// TwinCAT 3 PLC project dmms
// ProgramVersion: 3.1.4026.18
// libraries:
//   Tc2_Standard, * (Beckhoff Automation GmbH)
//   Tc2_System, * (Beckhoff Automation GmbH)
//   Tc3_Mc3PlanarMotion, * (Beckhoff Automation GmbH)
//   Tc3_Physics, * (Beckhoff Automation GmbH)
//   Tc3_XPlanarStandard, * (Beckhoff Automation GmbH)
//   Tc3_XPlanarUtility, * (Beckhoff Automation GmbH)
// project tree:
//   / PlcTask.TcTTO
//   POUs/ FB_MotionSystem.TcPOU, MAIN.TcPOU

CONFIGURATION dmms
    RESOURCE PLC ON TwinCAT3
        TASK PlcTask(INTERVAL := T#10ms, PRIORITY := 21);
        PROGRAM MAIN WITH PlcTask : MAIN;
    END_RESOURCE
END_CONFIGURATION

// ---- POUs/MAIN.TcPOU
PROGRAM MAIN
VAR
	fbXMotionUnit : FB_MotionSystem;
	nState : UDINT;
END_VAR

CASE nState OF
	0: // Init
		nState := nState + 1;
	1: // Startup sequence
		IF fbXMotionUnit.Startup() THEN
			nState := nState + 29;
		END_IF
	30: // Preparing sequence
		IF fbXMotionUnit.Starting(bReset:= FALSE) THEN
			nState := nState + 10;
		END_IF
	40: // Executing sequence
		fbXMotionUnit.Execute(bReset:= FALSE);
END_CASE
// Cyclic update
fbXMotionUnit.Cycle();

END_PROGRAM

// ---- POUs/FB_MotionSystem.TcPOU
FUNCTION_BLOCK FB_MotionSystem
VAR
	fbXPlanarSystem : FB_XPlanarSystem;
	fbXPlanarMover  : ARRAY[1..maxNumMover] OF FB_XPlanarMoverStandard;
	nStartupSequence   : UDINT;
	nStartingSequence  : UDINT;
	nExecutingSequence : UDINT;
END_VAR

METHOD Cycle
VAR
    i : UDINT;
END_VAR
// Cyclic XPlanar objects update
fbXPlanarSystem.Cycle();
FOR i := 1 TO moverCount DO
fbXPlanarMover[i].Cycle();
END_FOR
END_METHOD

METHOD Execute : BOOL
VAR_INPUT
	bReset : BOOL; // Reset sequence
END_VAR
VAR
	i : UDINT;
END_VAR
VAR_INST
	targetPos    : ARRAY[1..maxNumMover] OF PositionXYC;
	bMoversInPos : BOOL;
	bMoverError  : BOOL;
END_VAR
IF bReset THEN
	Execute := FALSE;
	nExecutingSequence := 0;
END_IF

CASE nExecutingSequence OF
	0: // Init
		bMoversInPos := FALSE;
		bMoverError := FALSE;
		IF NOT bReset THEN
			IF fbXPlanarMover[1].P_CommandMode = MC_PLANAR_MOVER_COMMAND_MODE.FreeMovement THEN
				nExecutingSequence := nExecutingSequence + 10;
			END_IF
		END_IF

	10: // Mover 1 -> X120 Y120, Mover 2 -> X360 Y600, 500 mm/s
		targetPos[1].SetValuesXYC(120, 120, 0);
		targetPos[2].SetValuesXYC(360, 600, 0);
		FOR i := 1 TO moverCount DO
			fbXPlanarMover[i].MoveToPosition('Move to XY', targetPos[i], 500, 1250, 1250, 12500);
		END_FOR
		nExecutingSequence := nExecutingSequence + 1;

	11: // Movers moving
		bMoversInPos := TRUE;
		bMoverError := FALSE;
		FOR i := 1 TO moverCount DO
			bMoversInPos := bMoversInPos AND fbXPlanarMover[i].P_MoveToPosition.Done;
			bMoverError  := bMoverError  OR  fbXPlanarMover[i].P_MoveToPosition.Error;
		END_FOR
		IF bMoversInPos THEN
			nExecutingSequence := nExecutingSequence + 9;
		ELSIF bMoverError THEN
			nExecutingSequence := nExecutingSequence + 4;
		END_IF

	20: // Mover 1 -> X120 Y600, Mover 2 -> X360 Y120, 500 mm/s
		targetPos[1].SetValuesXYC(120, 600, 0);
		targetPos[2].SetValuesXYC(360, 120, 0);
		FOR i := 1 TO moverCount DO
			fbXPlanarMover[i].MoveToPosition('Move to XY', targetPos[i], 500, 1250, 1250, 12500);
		END_FOR
		nExecutingSequence := nExecutingSequence + 1;

	21: // Movers moving
		bMoversInPos := TRUE;
		bMoverError := FALSE;
		FOR i := 1 TO moverCount DO
			bMoversInPos := bMoversInPos AND fbXPlanarMover[i].P_MoveToPosition.Done;
			bMoverError  := bMoverError  OR  fbXPlanarMover[i].P_MoveToPosition.Error;
		END_FOR
		IF bMoversInPos THEN
			nExecutingSequence := nExecutingSequence + 9;
		ELSIF bMoverError THEN
			nExecutingSequence := nExecutingSequence + 4;
		END_IF

	30: // Done - loop
		Execute := FALSE; // operator przerywa ręcznie (Stop / E-Stop)
		nExecutingSequence := nExecutingSequence - 20; // wraca do 10 - pętla
END_CASE
END_METHOD

METHOD Starting : BOOL
VAR_INPUT
	bReset : BOOL;
END_VAR
VAR
	i : UDINT;
END_VAR
VAR_INST
	// --- diagnostyka bledu enable ---
	nErrorID       : UDINT;    // surowy kod bledu
	sErrorHex      : STRING;   // ten sam kod w HEX (do szukania w InfoSys)
	nErrObjType    : UDINT;    // typ obiektu, ktory zawinil
	nErrObjID      : UDINT;    // ktory konkretnie (np. mover 2)
	stStartCheck   : ARRAY[1..maxNumMover] OF ST_CheckStartConditionFeedback;  // czemu pozycja zla
END_VAR
IF bReset THEN
	Starting := FALSE;
	nStartingSequence := 0;
END_IF

CASE nStartingSequence OF
	0: // Init
		Execute(bReset := TRUE);
		IF NOT bReset THEN
			nStartingSequence := nStartingSequence + 50;   // -> 50
		END_IF

	50: // Enable movers command
		IF fbXPlanarSystem.EnableMovers() THEN
			nStartingSequence := nStartingSequence + 1;    // -> 51
		END_IF

	51: // Enabling movers
		IF fbXPlanarSystem.P_EnableMovers.Done THEN
			nStartingSequence := nStartingSequence + 29;   // -> 80 (OK)
				ELSIF fbXPlanarSystem.P_EnableMovers.Error THEN
			nErrorID    := fbXPlanarSystem.P_EnableMovers.ErrorID;
			nErrObjType := fbXPlanarSystem.P_EnableMovers.stInfo.nObjectType;
			nErrObjID   := fbXPlanarSystem.P_EnableMovers.stInfo.nObjectID;
			FOR i := 1 TO moverCount DO
				stStartCheck[i] := fbXPlanarMover[i].CheckStartConditions();
			END_FOR
			nStartingSequence := nStartingSequence + 4;    // -> 55 (blad)
		END_IF

	55: // Enable movers FAILED - stoimy tu; wszystkie dane bledu w zmiennych powyzej
		;

	80: // Done
		Starting := TRUE;
END_CASE
END_METHOD

METHOD Startup : BOOL
VAR
	i : UDINT;
END_VAR
CASE nStartupSequence OF
	0: // Init
		nStartupSequence := nStartupSequence + 1;
	1: // Assign mover references to the system
	FOR i := 1 TO moverCount DO
		fbXPlanarSystem.SetMoverStandard(i, fbXPlanarMover[i]);
	END_FOR
	nStartupSequence := nStartupSequence + 29;
	30: // Done
	Startup := TRUE;
END_CASE
END_METHOD

END_FUNCTION_BLOCK
